(* IEC 61131-3 sources: AXOpen/src/components.abstractions/ctrl/src, 4 files *)

(* ---- AxoDictionaryIdentifier.st ---- *)
NAMESPACE AXOpen.Components.Abstractions
    TYPE AxoDictionaryIdentifier :
        STRUCT
            Id    :   UINT;
        END_STRUCT;
    END_TYPE
END_NAMESPACE

(* ---- IAxoCodeReader.st ---- *)
USING AXOpen.Core;
NAMESPACE AXOpen.Components.Abstractions
    INTERFACE PUBLIC IAxoCodeReader
        METHOD ClearResultData : IAxoTaskState END_METHOD
        METHOD Read : IAxoTaskState
            VAR_OUTPUT
                result : ARRAY [0..245] OF BYTE;
            END_VAR
        END_METHOD
    END_INTERFACE
END_NAMESPACE

(* ---- IAxoVisionSensor.st ---- *)
USING AXOpen.Core;
NAMESPACE AXOpen.Components.Abstractions
    INTERFACE PUBLIC IAxoVisionSensor
        METHOD ClearInspectionResults : IAxoTaskState END_METHOD
        METHOD Trigger : IAxoTaskState END_METHOD
        METHOD ChangeJob : IAxoTaskState  VAR_INPUT Job : UINT; END_VAR END_METHOD
        METHOD ChangeJob : IAxoTaskState  VAR_INPUT Job : STRING; END_VAR END_METHOD
    END_INTERFACE
END_NAMESPACE

(* ---- AxoComponent_Status.st ---- *)
USING AXOpen.Core;

NAMESPACE AXOpen.Components.Abstractions
    {#ix-attr:[Container(Layout.Stack)]}
    {S7.extern=ReadWrite}
    CLASS PUBLIC AxoComponent_Status
        VAR PUBLIC
            {#ix-set:AttributeName = "ActionDescription: |[[1]ActionDescription]|"}
            {#ix-attr:[WarningLevel(500)]}
            {#ix-attr:[ErrorLevel(700)]}
            Action    :   AXOpen.Core.AxoTextList;
            {#ix-set:AttributeName = "ErrorDescription: |[[1]ErrorDescription]|"}
            {#ix-attr:[WarningLevel(500)]}
            {#ix-attr:[ErrorLevel(700)]}
            Error     :   AXOpen.Core.AxoTextList;
        END_VAR
    END_CLASS
END_NAMESPACE
